FUNCTION_BLOCK FB_Actuator EXTENDS FB_Device
VAR_INPUT
	cmd					: E_ActuatorCommand := E_ActuatorCommand.None;
	
	inpHome				AT %I* : BOOL;
	inpWork				AT %I* : BOOL;
END_VAR
VAR_OUTPUT
	stsState			: E_ActuatorState := E_ActuatorState.AtHome;
	stsFaultCode		: DINT;
	
	outHome				AT %Q* : BOOL;
	outWork				AT %Q* : BOOL;
END_VAR
VAR
	WorkTimer			: TON;
	HomeTimer			: TON;
	WorkSimTime			: TIME := T#2S;
	HomeSimTime			: TIME := T#2S;
	WorkFailTime		: TIME := T#10S;
	HomeFailTime		: TIME := T#10S;
END_VAR

Faults();
StateMachine();
Control();

METHOD Control : BOOL
VAR_INPUT
END_VAR
outHome := stsState = (E_ActuatorState.AtHome OR E_ActuatorState.GoingToHome);
outWork := stsState = (E_ActuatorState.AtWork OR E_ActuatorState.GoingToWork);
END_METHOD

METHOD Faults : BOOL
VAR_INPUT
END_VAR
WorkTimer(IN := stsState = E_ActuatorState.GoingToWork, PT := WorkFailTime);
HomeTimer(IN := stsState = E_ActuatorState.GoingToHome, PT := HomeFailTime);
IF WorkTimer.Q THEN
	stsFaultCode := 100;
ELSIF HomeTImer.Q THEN
	stsFaultCode := 200;
ELSE
	stsFaultCode := 0;
END_IF
END_METHOD

METHOD Simulate : BOOL
VAR_INPUT
END_VAR
inpWork := outWork AND WorkTimer.ET >= WorkSimTime;
inpHome := outHome AND HomeTimer.ET >= HomeSimTime;
END_METHOD

METHOD StateMachine : BOOL
VAR_INPUT
END_VAR
IF inpSim THEN
	Simulate();
END_IF

CASE stsState OF
	E_ActuatorState.AtHome:
		IF cmd = E_ActuatorCommand.Work THEN
			stsState := E_ActuatorState.GoingToWork;
		END_IF
	E_ActuatorState.AtWork:
		IF cmd = E_ActuatorCommand.Home THEN
			stsState := E_ActuatorState.GoingToHome;
		END_IF
	E_ActuatorState.GoingToHome:
		IF inpHome THEN
			stsState := E_ActuatorState.AtHome;
		ELSIF cmd = E_ActuatorCommand.Work THEN
			stsState := E_ActuatorState.GoingToWork;
		END_IF
	E_ActuatorState.GoingToWork:
		IF inpWork THEN
			stsState := E_ActuatorState.AtWork;
		ELSIF cmd = E_ActuatorCommand.Home THEN
			stsState := E_ActuatorState.GoingToHome;
		END_IF
END_CASE
END_METHOD

END_FUNCTION_BLOCK

(* stored: Version 1.1.0.1, ProductVersion 3.1.4024.4
   POU FB_Actuator: Id {3cd68f66-e8c0-4a60-9389-8668b3a2b172}, SpecialFunc None
   Method Control: Id {93764544-4736-43dc-9109-a4b0ef105662}
   Method Faults: Id {38735c76-907a-4ab6-8cce-b9e2ca074fec}
   Method Simulate: Id {0e859ce1-160c-4645-b9b6-f843fb29527f}
   Method StateMachine: Id {95e81728-9f5d-4f71-aa89-367478500cdc} *)
